{attribute 'qualified_only'}
VAR_GLOBAL
	eMode : E_Mode;
END_VAR

(* stored: Version 1.1.0.1, ProductVersion 3.1.4024.12
   GVL Output: Id {50a502ef-8b02-4dba-9ade-2130b92b9e72} *)
